(* Logix 5000 project; controller L3 vendor 1 type 14 code 92 rev 20.12; software revision 20.04; part 7 of 9 *)
(* tags used below, declared in another part *)
   A_CV_DEC_CH : REAL;
   A_CV_DEG : REAL;
   aux_dec_froid : REAL;
   aux_manu_dec_fr : REAL;
   auxtempfroiddec : DINT;
   B3 : DINT[100];
   chauffe_fort : BOOL;
   CONV_PID_N10_170 : PID;   // *** Tag created for conversion to PID type required for instruction translation ***
   CONV_PID_N10_50 : PID;   // *** Tag created for conversion to PID type required for instruction translation ***
   csg_fermet_v_Dec_froid : DINT;
   cv_ch_dec : REAL;
   DateTime : DINT[7];   // DINT array tag for retrieve wallclock time through GSV created during conversion
   delta_3min_dec : DINT;
   delta_sp_dec : DINT;
   F8 : REAL[100];
   kp_dec_ch : REAL;
   N10 : DINT[233];
   N7 : DINT[200];
   N9 : DINT[200];   // niveau decapage vers lancy (n9[10) ;;N9[70]
   offsetdecfrois : DINT;
   ok_dec_chauffe : BOOL;
   ok_dec_refroidir : BOOL;
   ons7 : BOOL;
   ons8 : BOOL;
   ons9 : BOOL;
   out_v_ch_dec : REAL;
   passage_jour_mois : BOOL;
   pid_dec_ch : PID;
   pid_dec_fr : PID;
   pid_deg : PID;
   refroidis_fort : BOOL;
   regul_anob : BOOL;
   S_BP_manu_DEC : BOOL;
   S_csg_manu_dec_ch : DINT;
   S_csg_manu_Dec_froid : DINT;
   s_pos_dec_ch : REAL;
   S_pos_dec_FR : REAL;
   S_RUN_PMP_DEC1 : BOOL;
   S_RUN_PMP_DEC2 : BOOL;
   S_SP_DEGRAIS : DINT;
   s_T_2_DEC : REAL;
   S_T_DEC : DINT;
   S_T_DEC2 : DINT;
   scp_CV_ch_dec : SCP;
   SCP_CV_DEC_CH : SCP;
   SCP_CV_DEG : SCP;
   scp_out_v_ch_dec : SCP;
   scp_pos_v_ch_dec : SCP;
   scp_pos_Vroid_dec : SCP;
   scp_t_2_dec : SCP;
   scp_Vanne_Vroid_dec : SCP;
   T4 : TIMER[180];
(* _2_GENERAL, continued *)

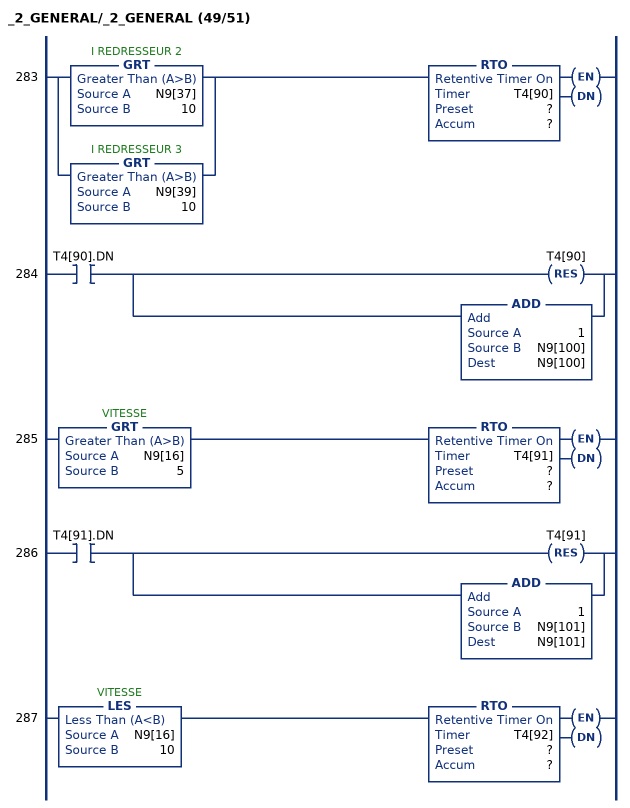
   283: [GRT(N9[37],10) ,GRT(N9[39],10) ]RTO(T4[90],?,?);
   284: XIC(T4[90].DN)[RES(T4[90]) ,ADD(1,N9[100],N9[100]) ];
   285: GRT(N9[16],5)RTO(T4[91],?,?);
   286: XIC(T4[91].DN)[RES(T4[91]) ,ADD(1,N9[101],N9[101]) ];
   287: LES(N9[16],10)RTO(T4[92],?,?);
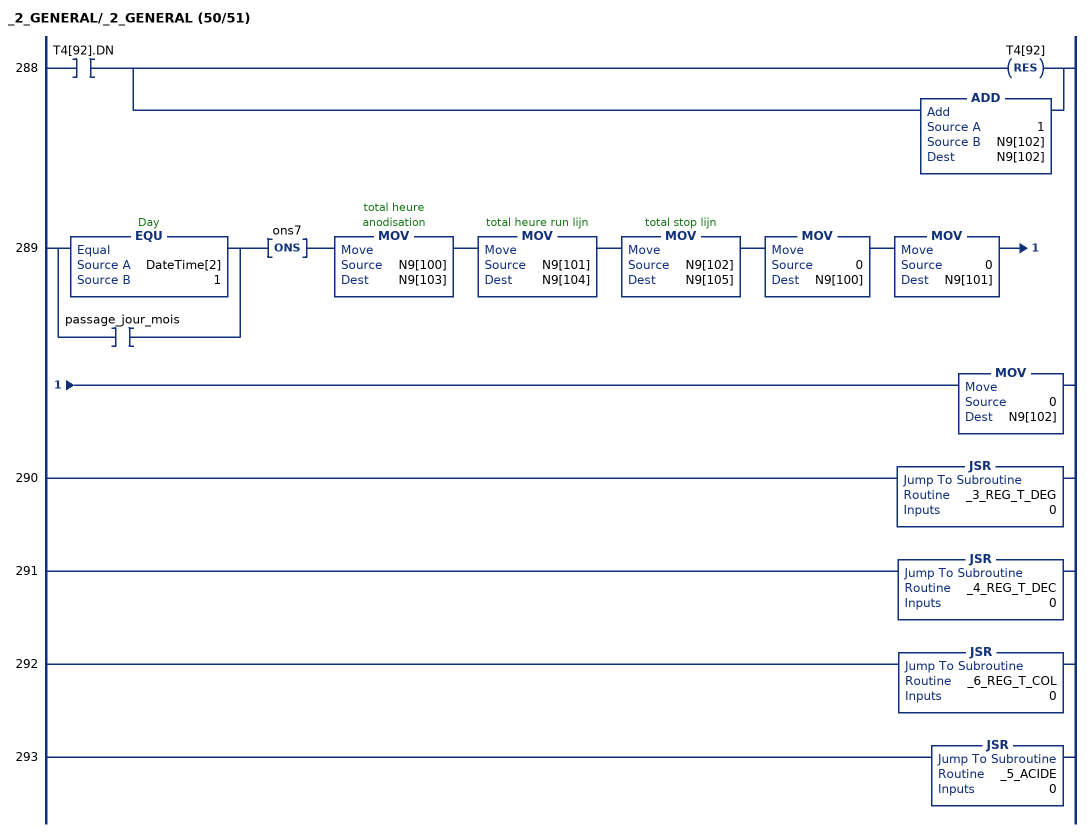
   288: XIC(T4[92].DN)[RES(T4[92]) ,ADD(1,N9[102],N9[102]) ];
   289: [EQU(DateTime[2],1) ,XIC(passage_jour_mois) ]ONS(ons7)MOV(N9[100],N9[103])MOV(N9[101],N9[104])MOV(N9[102],N9[105])MOV(0,N9[100])MOV(0,N9[101])MOV(0,N9[102]);
   290: JSR(_3_REG_T_DEG,0);
   291: JSR(_4_REG_T_DEC,0);
   292: JSR(_6_REG_T_COL,0);
   293: JSR(_5_ACIDE,0);
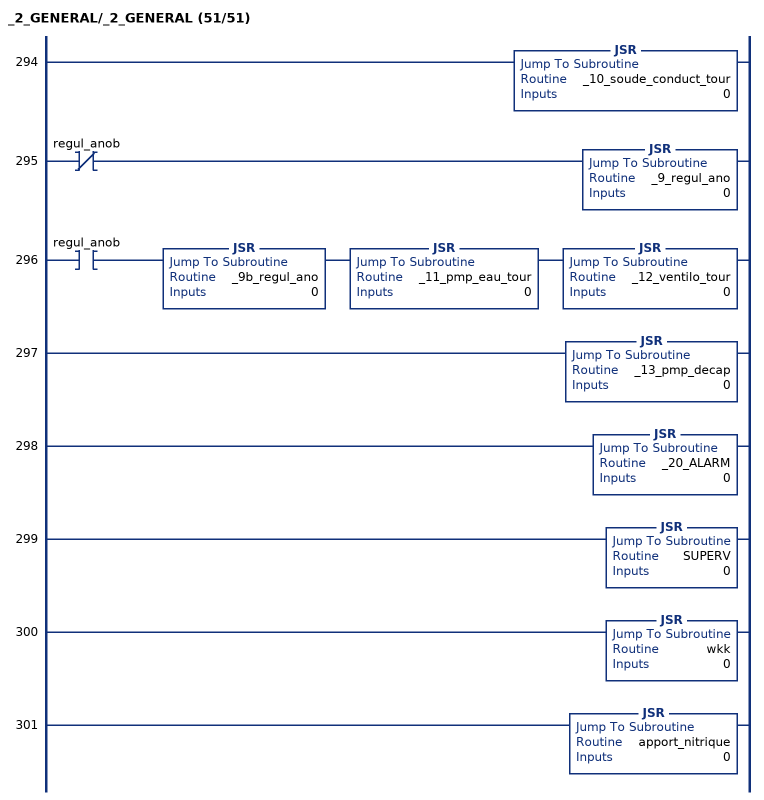
   294: JSR(_10_soude_conduct_tour,0);
   295: XIO(regul_anob)JSR(_9_regul_ano,0);
   296: XIC(regul_anob)JSR(_9b_regul_ano,0)JSR(_11_pmp_eau_tour,0)JSR(_12_ventilo_tour,0);
   297: JSR(_13_pmp_decap,0);
   298: JSR(_20_ALARM,0);
   299: JSR(SUPERV,0);
   300: JSR(wkk,0);
   301: JSR(apport_nitrique,0);
END_ROUTINE

ROUTINE _3_REG_T_DEG   (* ladder *)
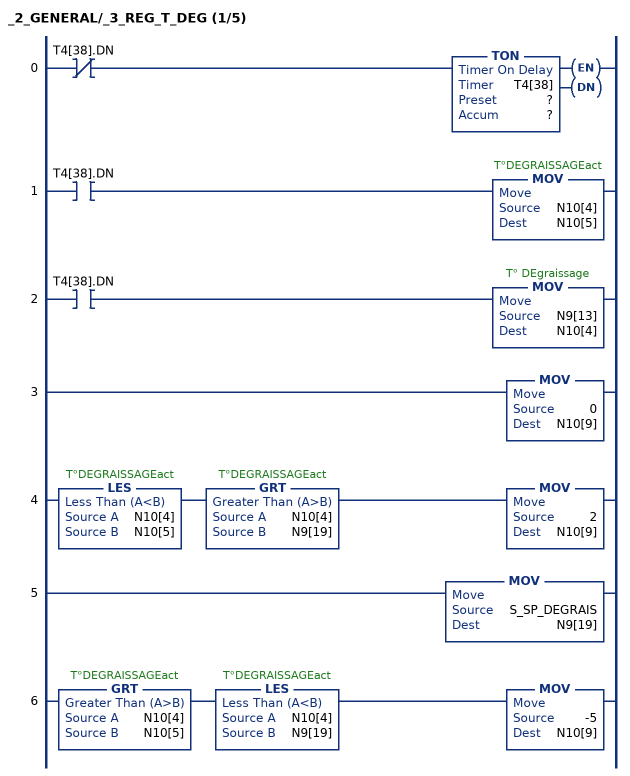
   0: XIO(T4[38].DN)TON(T4[38],?,?);
   1: XIC(T4[38].DN)MOV(N10[4],N10[5]);
   2: XIC(T4[38].DN)MOV(N9[13],N10[4]);
   3: MOV(0,N10[9]);
   4: LES(N10[4],N10[5])GRT(N10[4],N9[19])MOV(2,N10[9]);
   5: MOV(S_SP_DEGRAIS,N9[19]);
   6: GRT(N10[4],N10[5])LES(N10[4],N9[19])MOV(-5,N10[9]);
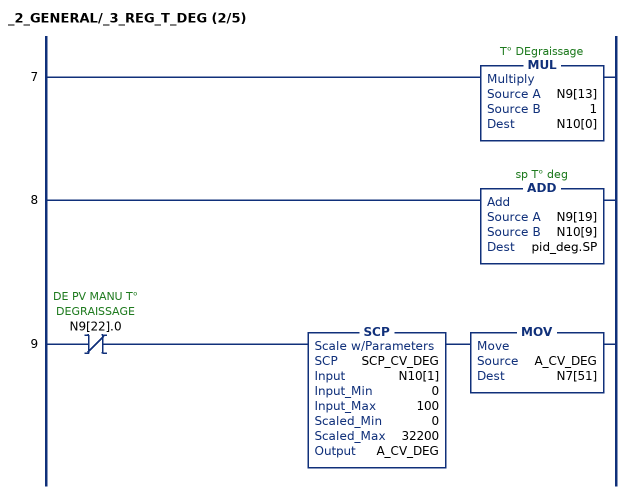
   7: MUL(N9[13],1,N10[0]);
   8: ADD(N9[19],N10[9],pid_deg.SP);
   9: XIO(N9[22].0)SCP(SCP_CV_DEG,N10[1],0,100,0,32200,A_CV_DEG)MOV(A_CV_DEG,N7[51]);
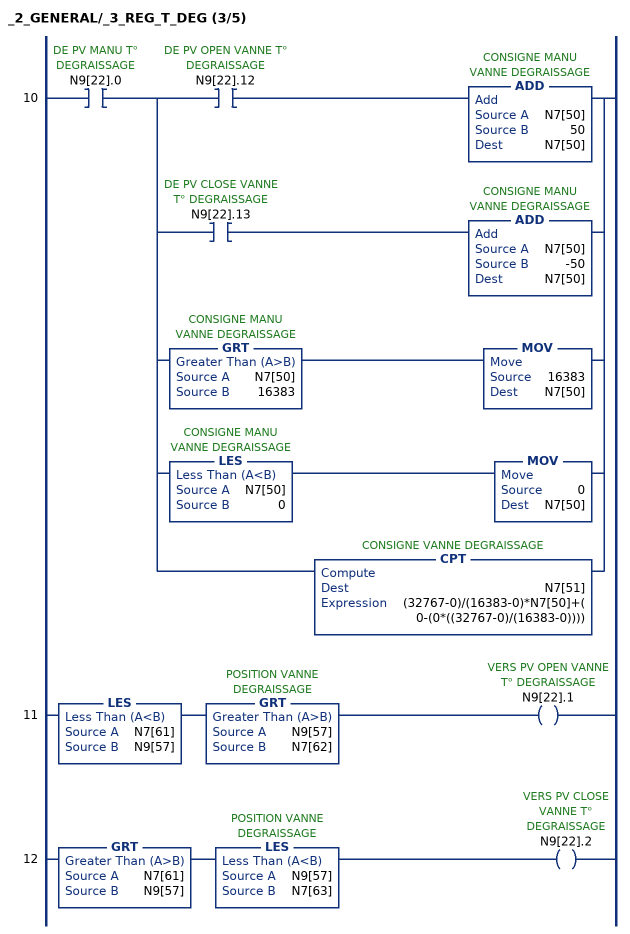
   10: XIC(N9[22].0)[XIC(N9[22].12) ADD(N7[50],50,N7[50]) ,XIC(N9[22].13) ADD(N7[50],-50,N7[50]) ,GRT(N7[50],16383) MOV(16383,N7[50]) ,LES(N7[50],0) MOV(0,N7[50]) ,CPT(N7[51],(32767-0)/(16383-0)*N7[50]+(0-(0*((32767-0)/(16383-0))))) ];
   11: LES(N7[61],N9[57])GRT(N9[57],N7[62])OTE(N9[22].1);
   12: GRT(N7[61],N9[57])LES(N9[57],N7[63])OTE(N9[22].2);
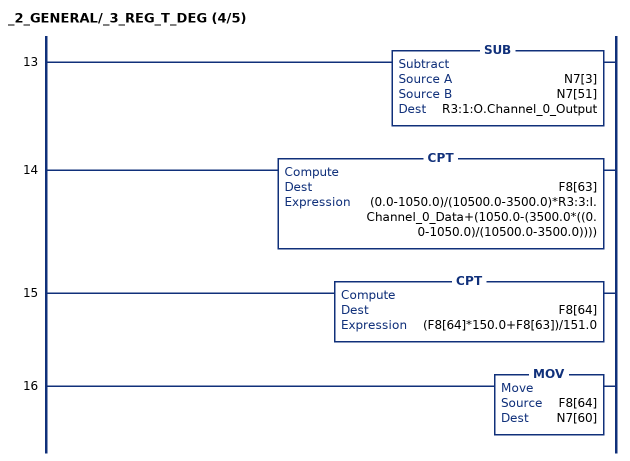
   13: SUB(N7[3],N7[51],R3:1:O.Channel_0_Output);
   14: CPT(F8[63],(0.0-1050.0)/(10500.0-3500.0)*R3:3:I.Channel_0_Data+(1050.0-(3500.0*((0.0-1050.0)/(10500.0-3500.0)))));
   15: CPT(F8[64],(F8[64]*150.0+F8[63])/151.0);
   16: MOV(F8[64],N7[60]);
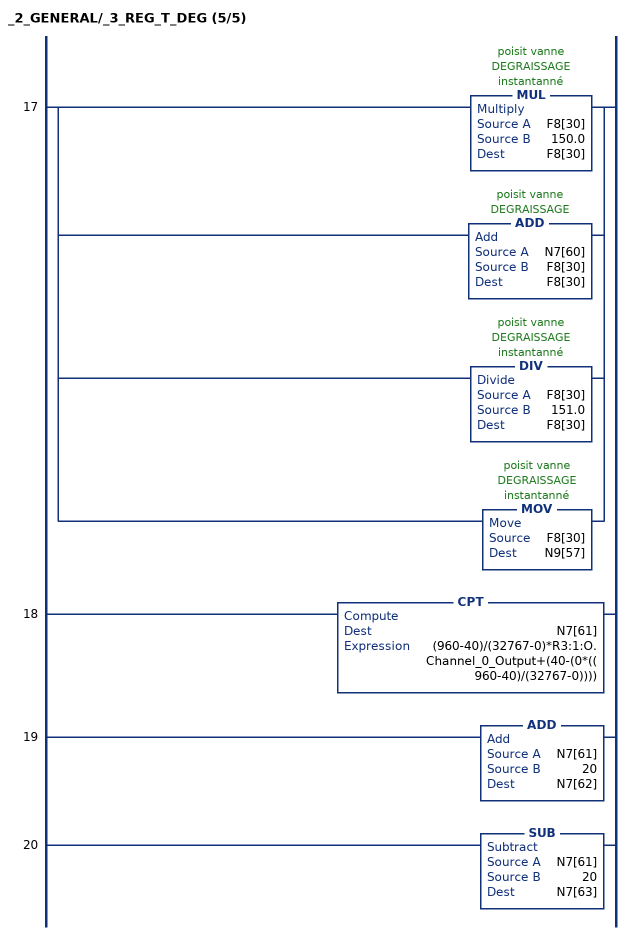
   17: [MUL(F8[30],150.0,F8[30]) ,ADD(N7[60],F8[30],F8[30]) ,DIV(F8[30],151.0,F8[30]) ,MOV(F8[30],N9[57]) ];
   18: CPT(N7[61],(960-40)/(32767-0)*R3:1:O.Channel_0_Output+(40-(0*((960-40)/(32767-0)))));
   19: ADD(N7[61],20,N7[62]);
   20: SUB(N7[61],20,N7[63]);
END_ROUTINE

ROUTINE _4_REG_T_DEC   (* ladder *)
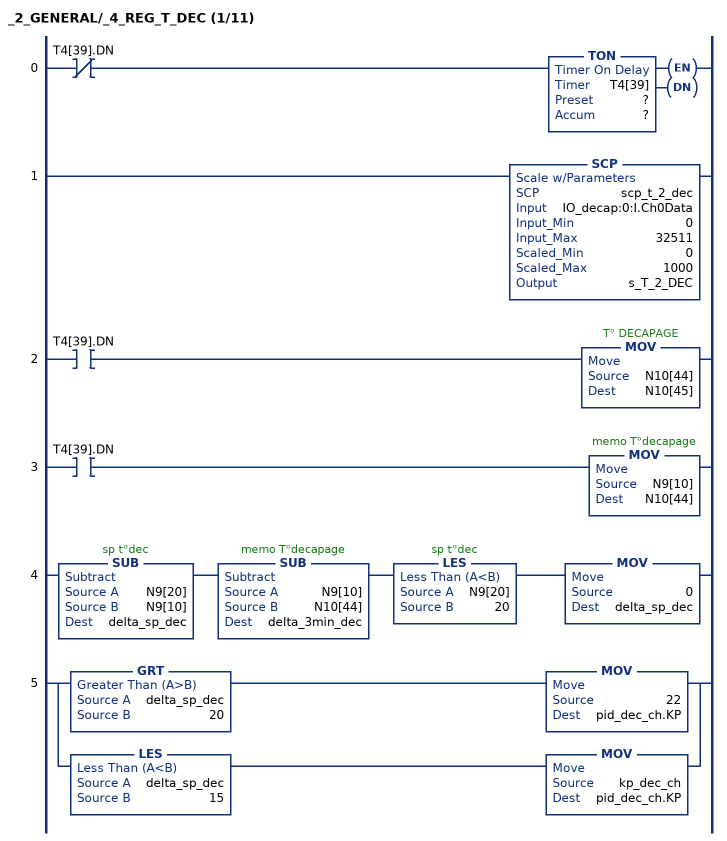
   0: XIO(T4[39].DN)TON(T4[39],?,?);
   1: SCP(scp_t_2_dec,IO_decap:0:I.Ch0Data,0,32511,0,1000,s_T_2_DEC);
   2: XIC(T4[39].DN)MOV(N10[44],N10[45]);
   3: XIC(T4[39].DN)MOV(N9[10],N10[44]);
   4: SUB(N9[20],N9[10],delta_sp_dec)SUB(N9[10],N10[44],delta_3min_dec)LES(N9[20],20)MOV(0,delta_sp_dec);
   5: [GRT(delta_sp_dec,20) MOV(22,pid_dec_ch.KP) ,LES(delta_sp_dec,15) MOV(kp_dec_ch,pid_dec_ch.KP) ];
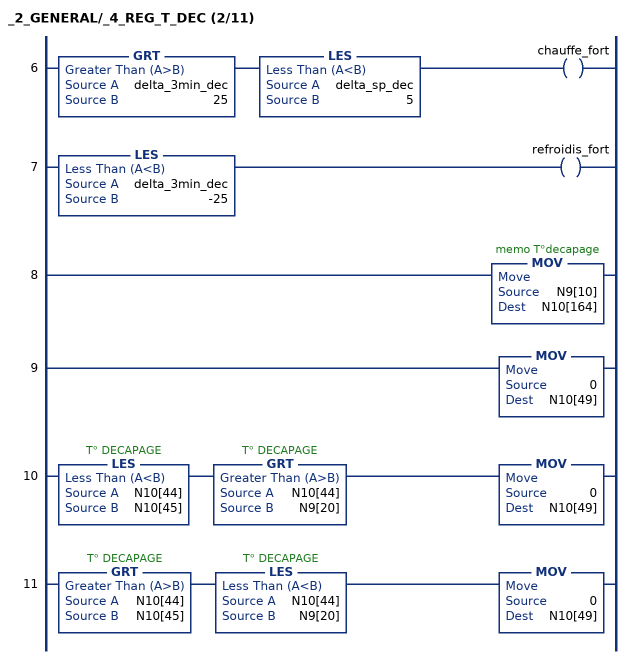
   6: GRT(delta_3min_dec,25)LES(delta_sp_dec,5)OTE(chauffe_fort);
   7: LES(delta_3min_dec,-25)OTE(refroidis_fort);
   8: MOV(N9[10],N10[164]);
   9: MOV(0,N10[49]);
   10: LES(N10[44],N10[45])GRT(N10[44],N9[20])MOV(0,N10[49]);
   11: GRT(N10[44],N10[45])LES(N10[44],N9[20])MOV(0,N10[49]);
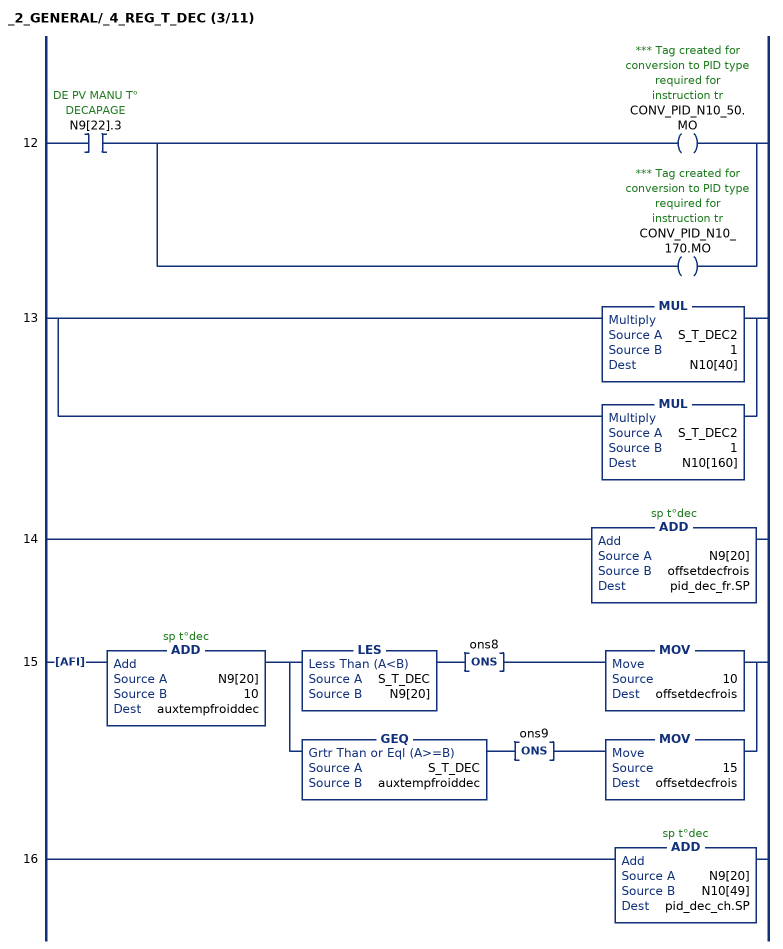
   12: XIC(N9[22].3)[OTE(CONV_PID_N10_50.MO) ,OTE(CONV_PID_N10_170.MO) ];
   13: [MUL(S_T_DEC2,1,N10[40]) ,MUL(S_T_DEC2,1,N10[160]) ];
   14: ADD(N9[20],offsetdecfrois,pid_dec_fr.SP);
   15: AFI()ADD(N9[20],10,auxtempfroiddec)[LES(S_T_DEC,N9[20]) ONS(ons8) MOV(10,offsetdecfrois) ,GEQ(S_T_DEC,auxtempfroiddec) ONS(ons9) MOV(15,offsetdecfrois) ];
   16: ADD(N9[20],N10[49],pid_dec_ch.SP);
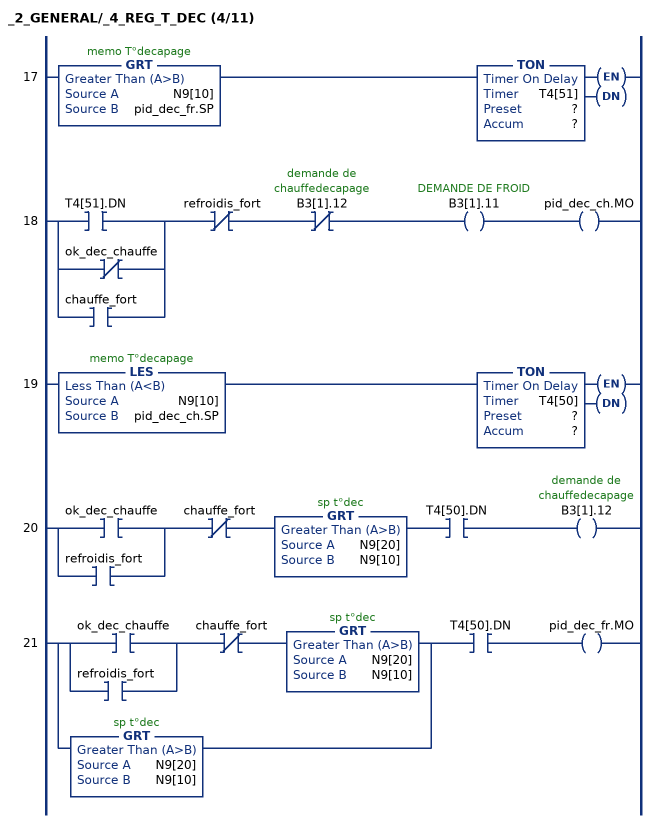
   17: GRT(N9[10],pid_dec_fr.SP)TON(T4[51],?,?);
   18: [XIC(T4[51].DN) ,XIO(ok_dec_chauffe) ,XIC(chauffe_fort) ]XIO(refroidis_fort)XIO(B3[1].12)OTE(B3[1].11)OTE(pid_dec_ch.MO);
   19: LES(N9[10],pid_dec_ch.SP)TON(T4[50],?,?);
   20: [XIC(ok_dec_chauffe) ,XIC(refroidis_fort) ]XIO(chauffe_fort)GRT(N9[20],N9[10])XIC(T4[50].DN)OTE(B3[1].12);
   21: [[XIC(ok_dec_chauffe) ,XIC(refroidis_fort) ] XIO(chauffe_fort) GRT(N9[20],N9[10]) ,GRT(N9[20],N9[10]) ]XIC(T4[50].DN)OTE(pid_dec_fr.MO);
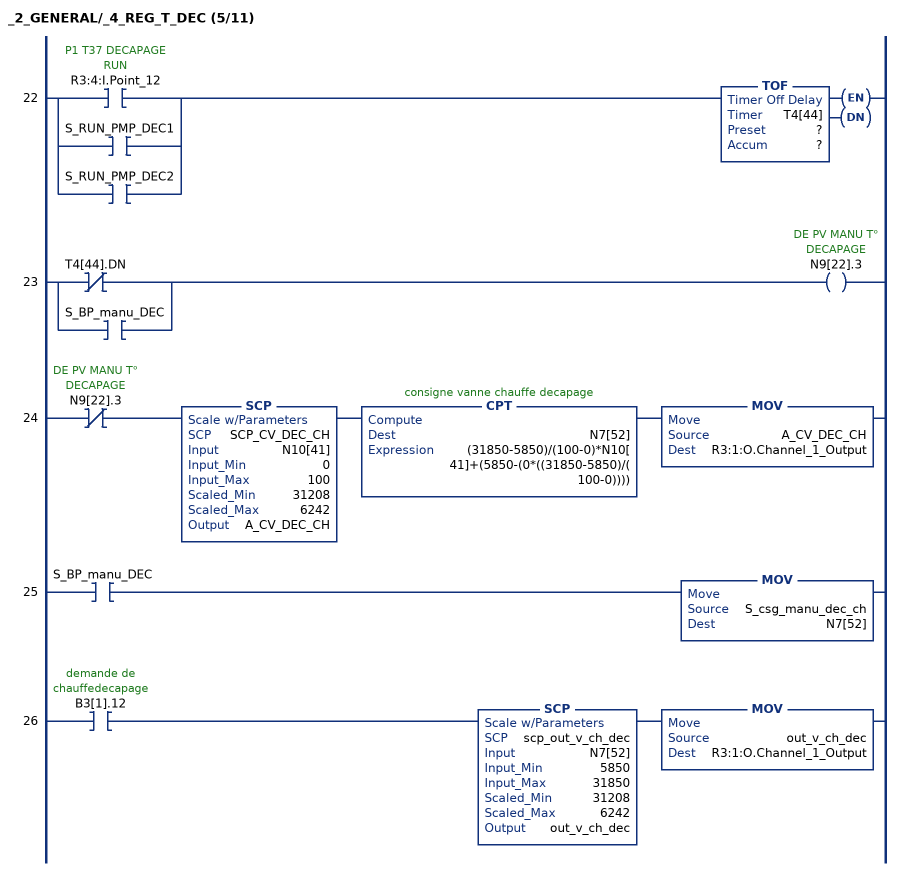
   22: [XIC(R3:4:I.Point_12) ,XIC(S_RUN_PMP_DEC1) ,XIC(S_RUN_PMP_DEC2) ]TOF(T4[44],?,?);
   23: [XIO(T4[44].DN) ,XIC(S_BP_manu_DEC) ]OTE(N9[22].3);
   24: XIO(N9[22].3)SCP(SCP_CV_DEC_CH,N10[41],0,100,31208,6242,A_CV_DEC_CH)CPT(N7[52],(31850-5850)/(100-0)*N10[41]+(5850-(0*((31850-5850)/(100-0)))))MOV(A_CV_DEC_CH,R3:1:O.Channel_1_Output);
   25: XIC(S_BP_manu_DEC)MOV(S_csg_manu_dec_ch,N7[52]);
   26: XIC(B3[1].12)SCP(scp_out_v_ch_dec,N7[52],5850,31850,31208,6242,out_v_ch_dec)MOV(out_v_ch_dec,R3:1:O.Channel_1_Output);
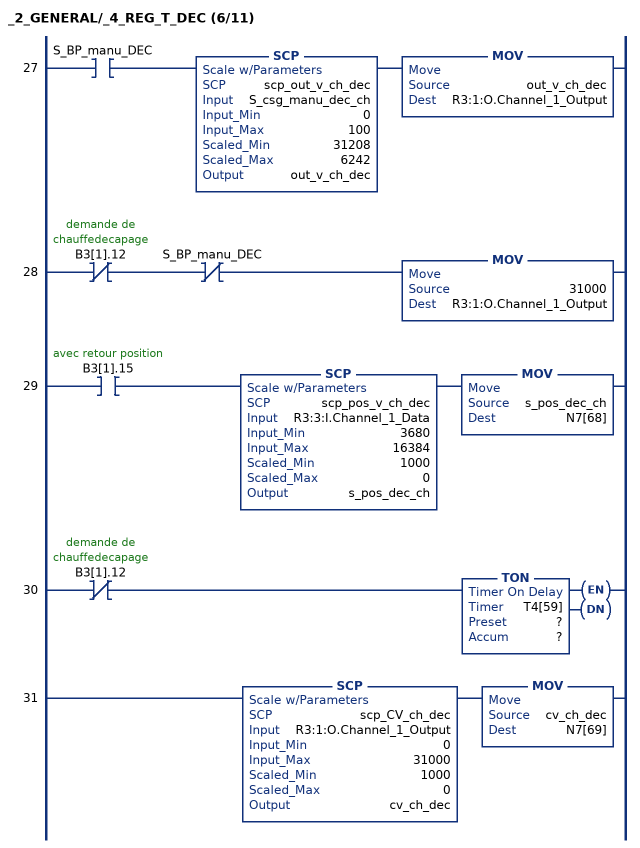
   27: XIC(S_BP_manu_DEC)SCP(scp_out_v_ch_dec,S_csg_manu_dec_ch,0,100,31208,6242,out_v_ch_dec)MOV(out_v_ch_dec,R3:1:O.Channel_1_Output);
   28: XIO(B3[1].12)XIO(S_BP_manu_DEC)MOV(31000,R3:1:O.Channel_1_Output);
   29: XIC(B3[1].15)SCP(scp_pos_v_ch_dec,R3:3:I.Channel_1_Data,3680,16384,1000,0,s_pos_dec_ch)MOV(s_pos_dec_ch,N7[68]);
   30: XIO(B3[1].12)TON(T4[59],?,?);
   31: SCP(scp_CV_ch_dec,R3:1:O.Channel_1_Output,0,31000,1000,0,cv_ch_dec)MOV(cv_ch_dec,N7[69]);
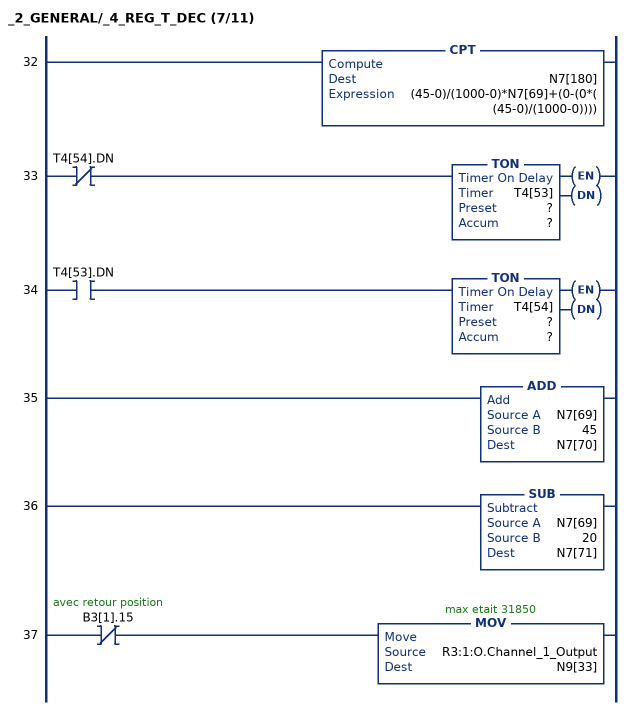
   32: CPT(N7[180],(45-0)/(1000-0)*N7[69]+(0-(0*((45-0)/(1000-0)))));
   33: XIO(T4[54].DN)TON(T4[53],?,?);
   34: XIC(T4[53].DN)TON(T4[54],?,?);
   35: ADD(N7[69],45,N7[70]);
   36: SUB(N7[69],20,N7[71]);
   37: XIO(B3[1].15)MOV(R3:1:O.Channel_1_Output,N9[33]);
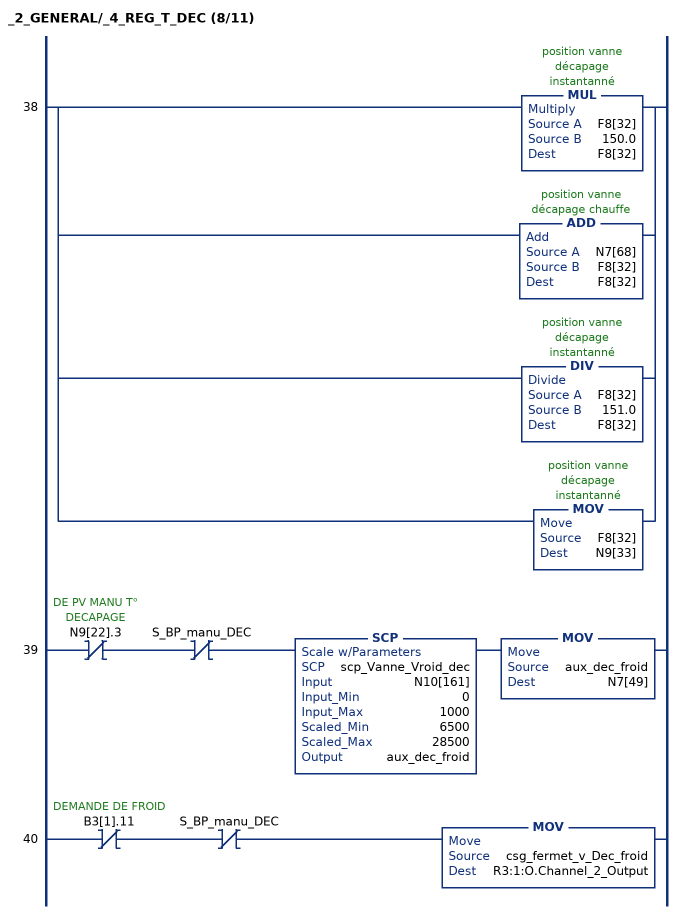
   38: [MUL(F8[32],150.0,F8[32]) ,ADD(N7[68],F8[32],F8[32]) ,DIV(F8[32],151.0,F8[32]) ,MOV(F8[32],N9[33]) ];
   39: XIO(N9[22].3)XIO(S_BP_manu_DEC)SCP(scp_Vanne_Vroid_dec,N10[161],0,1000,6500,28500,aux_dec_froid)MOV(aux_dec_froid,N7[49]);
   40: XIO(B3[1].11)XIO(S_BP_manu_DEC)MOV(csg_fermet_v_Dec_froid,R3:1:O.Channel_2_Output);
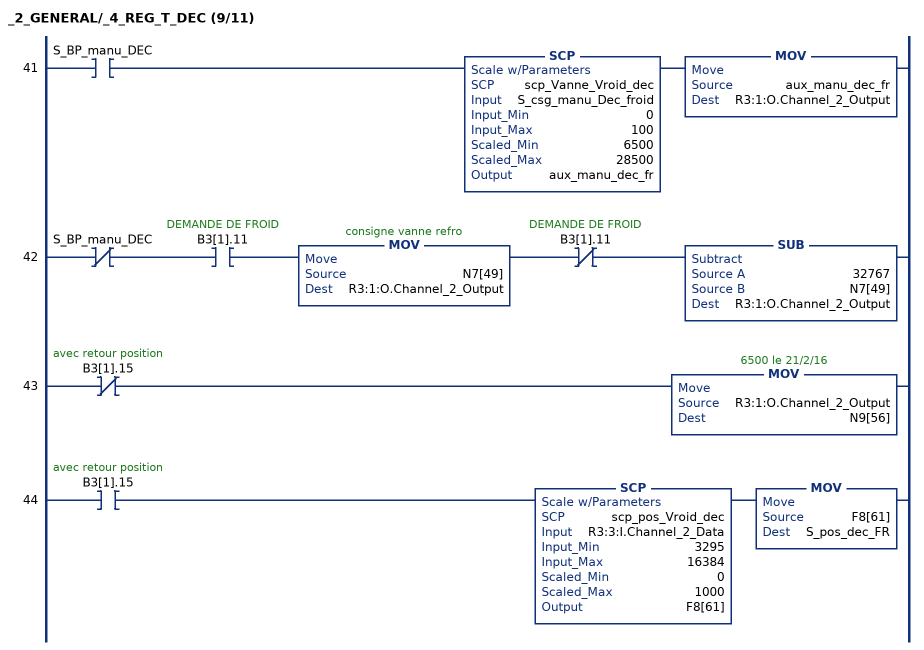
   41: XIC(S_BP_manu_DEC)SCP(scp_Vanne_Vroid_dec,S_csg_manu_Dec_froid,0,100,6500,28500,aux_manu_dec_fr)MOV(aux_manu_dec_fr,R3:1:O.Channel_2_Output);
   42: XIO(S_BP_manu_DEC)XIC(B3[1].11)MOV(N7[49],R3:1:O.Channel_2_Output)XIO(B3[1].11)SUB(32767,N7[49],R3:1:O.Channel_2_Output);
   43: XIO(B3[1].15)MOV(R3:1:O.Channel_2_Output,N9[56]);
   44: XIC(B3[1].15)SCP(scp_pos_Vroid_dec,R3:3:I.Channel_2_Data,3295,16384,0,1000,F8[61])MOV(F8[61],S_pos_dec_FR);
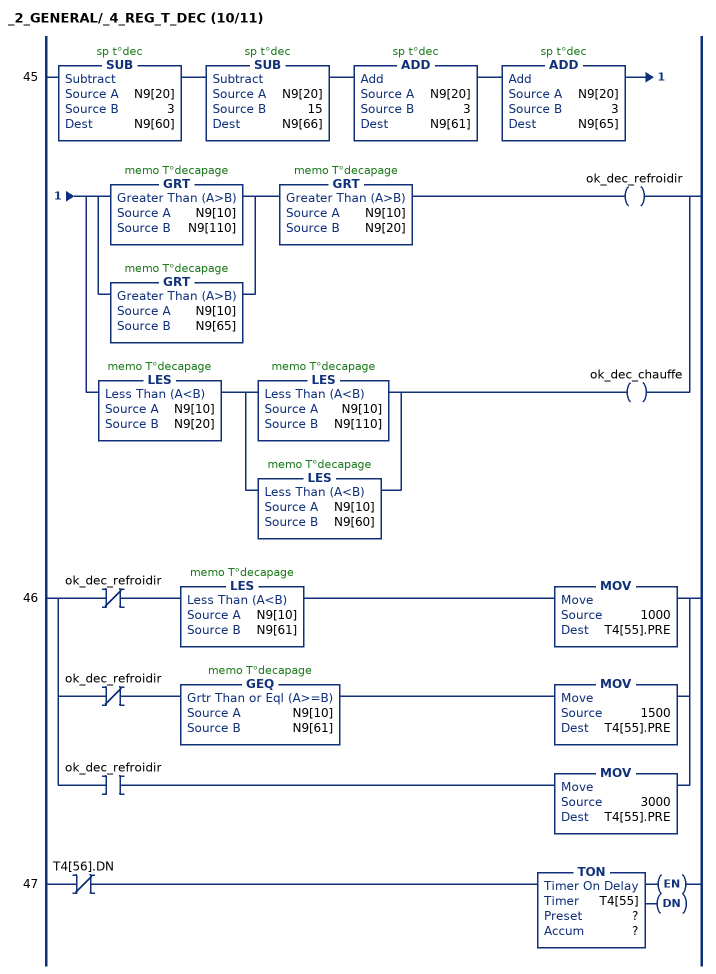
   45: SUB(N9[20],3,N9[60])SUB(N9[20],15,N9[66])ADD(N9[20],3,N9[61])ADD(N9[20],3,N9[65])[[GRT(N9[10],N9[110]) ,GRT(N9[10],N9[65]) ] GRT(N9[10],N9[20]) OTE(ok_dec_refroidir) ,LES(N9[10],N9[20]) [LES(N9[10],N9[110]) ,LES(N9[10],N9[60]) ] OTE(ok_dec_chauffe) ];
   46: [XIO(ok_dec_refroidir) LES(N9[10],N9[61]) MOV(1000,T4[55].PRE) ,XIO(ok_dec_refroidir) GEQ(N9[10],N9[61]) MOV(1500,T4[55].PRE) ,XIC(ok_dec_refroidir) MOV(3000,T4[55].PRE) ];
   47: XIO(T4[56].DN)TON(T4[55],?,?);
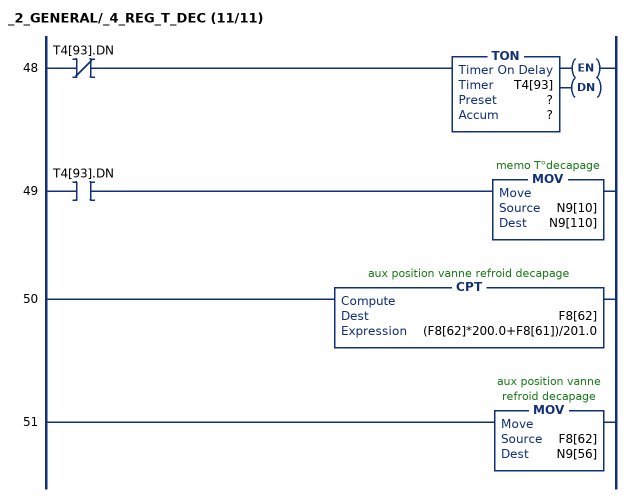
   48: XIO(T4[93].DN)TON(T4[93],?,?);
   49: XIC(T4[93].DN)MOV(N9[10],N9[110]);
   50: CPT(F8[62],(F8[62]*200.0+F8[61])/201.0);
   51: MOV(F8[62],N9[56]);
END_ROUTINE
